PROGRAM Stn052_PrgCalls
VAR
END_VAR

//Turn on the default programs
IF gFirstScan THEN
	gDebug_ComponentCalls.CallStn052_20_ReceivingBreakStopsGrn := TRUE;
	gDebug_ComponentCalls.CallStn052_21_ReceivingBreakStopsRed := TRUE;
	gDebug_ComponentCalls.CallStn052_35_Stn123Divert := TRUE;
	gDebug_ComponentCalls.CallStn052_36_Stn123MainMergePrestop := TRUE;
	gDebug_ComponentCalls.CallStn052_37_Stn123Merge := TRUE;
	gDebug_ComponentCalls.CallStn052_40_Stn124Divert := TRUE;
	gDebug_ComponentCalls.CallStn052_41_Stn124MainMergePrestop := TRUE;
	gDebug_ComponentCalls.CallStn052_42_Stn124Merge := TRUE;
	gDebug_ComponentCalls.CallStn052_45_Stn125Divert := TRUE;
	gDebug_ComponentCalls.CallStn052_46_Stn125MainMergePrestop := TRUE;
	gDebug_ComponentCalls.CallStn052_47_Stn125Merge := TRUE;
	gDebug_ComponentCalls.CallStn052_50_Stn126Divert := TRUE;
	gDebug_ComponentCalls.CallStn052_51_Stn126MainMergePrestop := TRUE;
	gDebug_ComponentCalls.CallStn052_52_Stn126Merge := TRUE;
END_IF

IF gDebug_ComponentCalls.CallStn052_20_ReceivingBreakStopsGrn OR
		gFirstScan THEN
	Stn052_20_ReceivingBreakStopsGrn();
END_IF
IF gDebug_ComponentCalls.CallStn052_21_ReceivingBreakStopsRed OR
		gFirstScan THEN	
	Stn052_21_ReceivingBreakStopsRed();
END_IF
IF gDebug_ComponentCalls.CallStn052_35_Stn123Divert OR
		gFirstScan THEN
	Stn052_35_Stn123Divert();
END_IF
IF gDebug_ComponentCalls.CallStn052_36_Stn123MainMergePrestop OR
		gFirstScan THEN	
	Stn052_36_Stn123MainMergePrestop();
END_IF
IF gDebug_ComponentCalls.CallStn052_37_Stn123Merge OR
		gFirstScan THEN	
	Stn052_37_Stn123Merge();
END_IF	
IF gDebug_ComponentCalls.CallStn052_40_Stn124Divert OR
		gFirstScan THEN	
	Stn052_40_Stn124Divert();
END_IF
IF gDebug_ComponentCalls.CallStn052_41_Stn124MainMergePrestop OR
		gFirstScan THEN	
	Stn052_41_Stn124MainMergePrestop();
END_IF	
IF gDebug_ComponentCalls.CallStn052_42_Stn124Merge OR
		gFirstScan THEN	
	Stn052_42_Stn124Merge();
END_IF	
IF gDebug_ComponentCalls.CallStn052_45_Stn125Divert OR
		gFirstScan THEN	
	Stn052_45_Stn125Divert();
END_IF	
IF gDebug_ComponentCalls.CallStn052_46_Stn125MainMergePrestop OR
		gFirstScan THEN	
	Stn052_46_Stn125MainMergePrestop();
END_IF
IF gDebug_ComponentCalls.CallStn052_47_Stn125Merge OR
		gFirstScan THEN	
	Stn052_47_Stn125Merge();
END_IF	
IF gDebug_ComponentCalls.CallStn052_50_Stn126Divert OR
		gFirstScan THEN	
	Stn052_50_Stn126Divert();
END_IF
IF gDebug_ComponentCalls.CallStn052_51_Stn126MainMergePrestop OR
		gFirstScan THEN	
	Stn052_51_Stn126MainMergePrestop();
END_IF
IF gDebug_ComponentCalls.CallStn052_52_Stn126Merge OR
		gFirstScan THEN	
	Stn052_52_Stn126Merge();
END_IF

END_PROGRAM

(* stored: Version 1.1.0.1, ProductVersion 3.1.4024.6
   POU Stn052_PrgCalls: Id {e99cef2f-b150-436d-98e7-c1b1c01fa284}, SpecialFunc None *)
